{region '#Template'}
	{attribute 'Version' := '1.0.0.0'}
	{attribute 'Tags' := '"LCID": "1031", "Text": "Types, Publisher, Subscriber, RA, Facade, Data"'}
	{attribute 'Tags' := '"LCID": "1033", "Text": "Types, Publisher, Subscriber, RA, Facade, Data"'}
	{attribute 'Description' := '"LCID": "1031", "Text": "Fassadendaten/-status für die Raumautomation"'}
	{attribute 'Description' := '"LCID": "1033", "Text": "Facade-data/-states for room-automation"'}
{endregion}
TYPE ST_BA_Facade :
STRUCT
		stSunBld 					: ST_BA_SunBld;	//  Telegram for					1)	burglary, fire, ice (building-wise)
													//					2)	storm-protection (calculated facade-wise)
													//					3)	Maintenance position (start- and adjustable for each facade)
													//					4)	facade-wise thermo-automation
													//					5)	facade-wise twilight-automation
													//					6)	facade-wise park-position
													
		bThAuto_Release				: BOOL;			// enable for the zone-wise thermo automatic
		bTwiLgtAuto_Release			: BOOL;			// enable for the zone-wise twilight automatic
		bSunPrtc_State				: BOOL;			// active-state from the facade-wise sun-protection-calculation (FB_BA_SunPrtc) -> further decisions have to be made in each zone
		fSunPrtc_Position			: REAL;			// position calculated by the facade-wise sun-protection-calculation (FB_BA_SunPrtc)
		fSunPrtc_Angle				: REAL;			// angle calculated by the facade-wise sun-protection-calculation (FB_BA_SunPrtc)
END_STRUCT
END_TYPE

(* stored: Version 1.1.0.1, ProductVersion 3.1.4024.9
   DUT ST_BA_Facade: Id {69298b8a-08ad-4112-a28a-ac2a67871f18} *)
